// TIA Portal V20 export
FUNCTION_BLOCK "FB_Visual_Test"   // FB7, LAD
{ S7_Optimized_Access := 'TRUE' }
// stored: MemoryReserve 100, SetENOAutomatically false
   VAR_INPUT
      Star_Functional_Test : Bool;
      Reset_Functional_Test : Bool;
      Button_Start_Approve : Bool;
      In_Test_Parameters : "IO_Device_Test_Parameters";
   END_VAR
   VAR_OUTPUT
      Visual_Test_Approved_PLC : Bool;
   END_VAR
   VAR
      Aux_Trigger : Bool;
      Timer_Delay_Start_Visual_Test { S7_SetPoint := 'True'} : TON_TIME;
      Timer_Delay_Reset { S7_SetPoint := 'True'} : TON_TIME;
   END_VAR
   VAR_TEMP   // added for the SCL form of the ladder/FBD networks
      _w1 : Bool;
   END_VAR
BEGIN

REGION Network 1
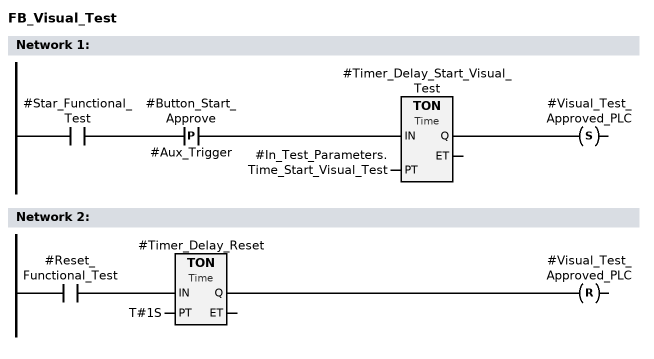
   RUNG wire#powerrail
      Contact( #Star_Functional_Test )
      P_Contact(operand := #Button_Start_Approve, bit := #Aux_Trigger)
      { S7_Templates := "time_type := Time" } #Timer_Delay_Start_Visual_Test.TON(pt := #In_Test_Parameters.Time_Start_Visual_Test, et =>)
      S_Coil( #Visual_Test_Approved_PLC )
   END_RUNG
   // the same network as SCL:
   #_w1 := #Star_Functional_Test AND #Button_Start_Approve AND NOT #Aux_Trigger;   // rising edge of #Button_Start_Approve
   #Aux_Trigger := #Button_Start_Approve;
   #Timer_Delay_Start_Visual_Test(IN := #_w1, PT := #In_Test_Parameters.Time_Start_Visual_Test);   // TON
   IF #Timer_Delay_Start_Visual_Test.Q THEN #Visual_Test_Approved_PLC := TRUE; END_IF;
END_REGION

REGION Network 2
   RUNG wire#powerrail
      Contact( #Reset_Functional_Test )
      { S7_Templates := "time_type := Time" } #Timer_Delay_Reset.TON(pt := T#1S, et =>)
      R_Coil( #Visual_Test_Approved_PLC )
   END_RUNG
   // the same network as SCL:
   #Timer_Delay_Reset(IN := #Reset_Functional_Test, PT := T#1S);   // TON
   IF #Timer_Delay_Reset.Q THEN #Visual_Test_Approved_PLC := FALSE; END_IF;
END_REGION
END_FUNCTION_BLOCK
